      CALL #s_TRS5_FB_HW_MTR_MS (
           i_CMD_Send_Stat          := #i_Send_Statistics,
           i_Event_DB               := "DB_Event_Section",
           i_Available_IO           := #i_IO_Available,
           i_IO_MS_Automatic_Mode   := TRUE,
           i_IO_NOT_THO             := #i_TRS5_IO_NOT_THO,
           i_CMD_Reset              := #i_CMD_Reset,
           i_CMD_Req_Motor_Forward  := #s_TRS5_Req_MTR_Run,
           i_CMD_Manual_Mode        := #i_Command.Manual,
           i_CMD_Manual_Run         := #i_Command.Man_TRS5_Start,
           o_IO_MTR                 := #o_TRS5_IO_MTR,
           o_ST_THO                 := #s_TRS5_ST_THO);

NETWORK
TITLE =PA: Tracking report TRS5
//Case 1: SCZ01 in position Straight
//- Direction Taken 2, Decision Level 8 with ID of TRS5
//
//Case 2: SCZ01 in position Down
//- Direction Taken 2, Decision Level 3 with ID of TRS2
//- Direction From 1, Decision Level 3 with ID of TRS5
//
//In position down.
//When the item entering the downstream section a message "Direction From" with
//value "1" is sent to HLC with The ID of the TRS5.
      NOP   0;
// Tracking report Direction to: 2 (Item goes from up to down) second message
      A     #s_TRS5_Send_Track_Report;
      FN    #s_TRS5_FN_Send_Track_Rep;
      JCN   PA06;

      A     #s_SWS1_ST_Down;
      JCN   PA04;

// Create reply route record if not existing
      CALL "FC_Read_Int_Record" (
           i_Record_Number          := #s_TRS5_Fnd_LNK,
           i_P_INT_Record           := "DB_UDT_LNK_Record".Rep_Route,
           i_DB                     := "DB_LNK_List",
           i_DB_Event_Num           := #t_DB_Event_Section_Num,
           o_INT                    := #s_TRS5_Rep_Route_Record);

      L     #s_TRS5_Rep_Route_Record;
      L     0;
      <=I   ;
      JCN   PA01;

      CALL "FC_Generator_LNK" (
           i_LNK                    := #s_TRS5_Fnd_LNK,
           i_DB_List                := #t_DB_Nr_Route_List,
           i_Default_Record         := -1,
           i_DB_Event_Num           := #t_DB_Event_Section_Num,
           o_LNK                    := #s_TRS5_Rep_Route_Record);

      CALL "FC_Read_Int_Record" (
           i_Record_Number          := #s_TRS5_Fnd_LNK,
           i_P_INT_Record           := "DB_UDT_LNK_Record".Rep_Route,
           i_DB                     := "DB_LNK_List",
           i_DB_Event_Num           := #t_DB_Event_Section_Num,
           o_INT                    := #s_TRS5_Rep_Route_Record);

      CALL "FC_Read_Int_Record" (
           i_Record_Number          := #s_TRS5_Fnd_LNK,
           i_P_INT_Record           := "DB_UDT_LNK_Record".LIC,
           i_DB                     := "DB_LNK_List",
           i_DB_Event_Num           := #t_DB_Event_Section_Num,
           o_INT                    := #t_LIC);

      CALL "FC_Read_ANY_Record" (
           i_Record_Number          := #t_LIC,
           i_ANY_Data_Record        := "DB_UDT_LIC_Record".BIR,
           i_ANY_Data               := "DB_Outgoing_Msgs".TrackingReport.Body.BIR,
           i_DB                     := "DB_LIC_List",
           i_DB_Event_Num           := #t_DB_Event_Section_Num);

      CALL "FC_Write_ANY_Record" (
           i_Record_Number          := #s_TRS5_Rep_Route_Record,
           i_ANY_Data_Record        := "DB_UDT_Route_Record".BIR,
           i_ANY_Data               := "DB_Outgoing_Msgs".TrackingReport.Body.BIR,
           i_DB                     := "DB_Route_List",
           i_DB_Event_Num           := #t_DB_Event_Section_Num);

// Update tracking report message
PA01: CALL "FC_Write_ANY_Record" (
           i_Record_Number          := #s_TRS5_Rep_Route_Record,
           i_ANY_Data_Record        := "DB_UDT_Route_Record".SuccessDirection,
           i_ANY_Data               := "DB_Route_List".Rep_Route[0].SuccessDirection,
           i_DB                     := "DB_Route_List",
           i_DB_Event_Num           := #t_DB_Event_Section_Num);

      CALL "FC_Write_Int_Record" (
           i_Record_Number          := #s_TRS5_Rep_Route_Record,
           i_P_INT_Record           := "DB_UDT_Route_Record".SuccessDirection.DirectionFrom,
           i_DB                     := "DB_Route_List",
           i_INT                    := 0,
           i_DB_Event_Num           := #t_DB_Event_Section_Num);

      CALL "FC_Write_Int_Record" (
           i_Record_Number          := #s_TRS5_Rep_Route_Record,
           i_P_INT_Record           := "DB_UDT_Route_Record".SuccessDirection.DirectionTaken,
           i_DB                     := "DB_Route_List",
           i_INT                    := 2,
           i_DB_Event_Num           := #t_DB_Event_Section_Num);

      CALL "FC_Write_Int_Record" (
           i_Record_Number          := #s_TRS5_Rep_Route_Record,
           i_P_INT_Record           := "DB_UDT_Route_Record".SuccessDirection.DecisionLevel,
           i_DB                     := "DB_Route_List",
           i_INT                    := 5,
           i_DB_Event_Num           := #t_DB_Event_Section_Num);

// Write sort report
      CALL "FC_Write_Event" (
           i_Message_ID             := 1201,//Tracking Report = 1201
           i_Event_value            := #s_TRS5_Fnd_LNK,
           i_DB_Event_Num           := #t_DB_Event_Section_Num,
           o_Return_Value           := #t_RET_VAL_int);
      JU    PA06;


// Tracking report Direction to: 2 (Item goes straight)
PA04: A     #s_SWS1_ST_Straight;
      JCN   PA06;

// Create reply route record if not existing
      CALL "FC_Read_Int_Record" (
           i_Record_Number          := #s_TRS5_Fnd_LNK,
           i_P_INT_Record           := "DB_UDT_LNK_Record".Rep_Route,
           i_DB                     := "DB_LNK_List",
           i_DB_Event_Num           := #t_DB_Event_Section_Num,
           o_INT                    := #s_TRS5_Rep_Route_Record);

      L     #s_TRS5_Rep_Route_Record;
      L     0;
      <=I   ;
      JCN   PA05;

      CALL "FC_Generator_LNK" (
           i_LNK                    := #s_TRS5_Fnd_LNK,
           i_DB_List                := #t_DB_Nr_Route_List,
           i_Default_Record         := -1,
           i_DB_Event_Num           := #t_DB_Event_Section_Num,
           o_LNK                    := #s_TRS5_Rep_Route_Record);

      CALL "FC_Read_Int_Record" (
           i_Record_Number          := #s_TRS5_Fnd_LNK,
           i_P_INT_Record           := "DB_UDT_LNK_Record".Rep_Route,
           i_DB                     := "DB_LNK_List",
           i_DB_Event_Num           := #t_DB_Event_Section_Num,
           o_INT                    := #s_TRS5_Rep_Route_Record);

      CALL "FC_Read_Int_Record" (
           i_Record_Number          := #s_TRS5_Fnd_LNK,
           i_P_INT_Record           := "DB_UDT_LNK_Record".LIC,
           i_DB                     := "DB_LNK_List",
           i_DB_Event_Num           := #t_DB_Event_Section_Num,
           o_INT                    := #t_LIC);

      CALL "FC_Read_ANY_Record" (
           i_Record_Number          := #t_LIC,
           i_ANY_Data_Record        := "DB_UDT_LIC_Record".BIR,
           i_ANY_Data               := "DB_Outgoing_Msgs".TrackingReport.Body.BIR,
           i_DB                     := "DB_LIC_List",
           i_DB_Event_Num           := #t_DB_Event_Section_Num);

      CALL "FC_Write_ANY_Record" (
           i_Record_Number          := #s_TRS5_Rep_Route_Record,
           i_ANY_Data_Record        := "DB_UDT_Route_Record".BIR,
           i_ANY_Data               := "DB_Outgoing_Msgs".TrackingReport.Body.BIR,
           i_DB                     := "DB_Route_List",
           i_DB_Event_Num           := #t_DB_Event_Section_Num);

// Update tracking report message
PA05: CALL "FC_Write_ANY_Record" (
           i_Record_Number          := #s_TRS5_Rep_Route_Record,
           i_ANY_Data_Record        := "DB_UDT_Route_Record".SuccessDirection,
           i_ANY_Data               := "DB_Route_List".Rep_Route[0].SuccessDirection,
           i_DB                     := "DB_Route_List",
           i_DB_Event_Num           := #t_DB_Event_Section_Num);

      CALL "FC_Write_Int_Record" (
           i_Record_Number          := #s_TRS5_Rep_Route_Record,
           i_P_INT_Record           := "DB_UDT_Route_Record".SuccessDirection.DirectionFrom,
           i_DB                     := "DB_Route_List",
           i_INT                    := 0,
           i_DB_Event_Num           := #t_DB_Event_Section_Num);

      CALL "FC_Write_Int_Record" (
           i_Record_Number          := #s_TRS5_Rep_Route_Record,
           i_P_INT_Record           := "DB_UDT_Route_Record".SuccessDirection.DirectionTaken,
           i_DB                     := "DB_Route_List",
           i_INT                    := 1,
           i_DB_Event_Num           := #t_DB_Event_Section_Num);

      CALL "FC_Write_Int_Record" (
           i_Record_Number          := #s_TRS5_Rep_Route_Record,
           i_P_INT_Record           := "DB_UDT_Route_Record".SuccessDirection.DecisionLevel,
           i_DB                     := "DB_Route_List",
           i_INT                    := 5,
           i_DB_Event_Num           := #t_DB_Event_Section_Num);

// Write sort report
      CALL "FC_Write_Event" (
           i_Message_ID             := 1201,//Tracking Report = 1201
           i_Event_value            := #s_TRS5_Fnd_LNK,
           i_DB_Event_Num           := #t_DB_Event_Section_Num,
           o_Return_Value           := #t_RET_VAL_int);

PA06: CALL #s_TRS5_FB_DAT (
           i_ID_Section             := #i_TRS5_ID,
           i_DB_Event               := "DB_Event_Section",
           i_PLC_Log_FIFO_DB        := "DB_LOG_Event_FIFO",
           i_CFG_BPI_Log_Level      := "DB_Setting".common.External_Log_Level,
           i_CFG_PLC_Log_Level      := "DB_Setting".common.Internal_Log_Level,
           i_CFG_PLC_Log_Route_Msgs := TRUE,
           i_CFG_PLC_LOG_BPI_Stat   := FALSE,
           i_CFG_PLC_No_Msg_To_Rout := #i_CFG_PLC_No_Msg_To_Rout);

NETWORK
TITLE =QA: Data layer of SCZ01
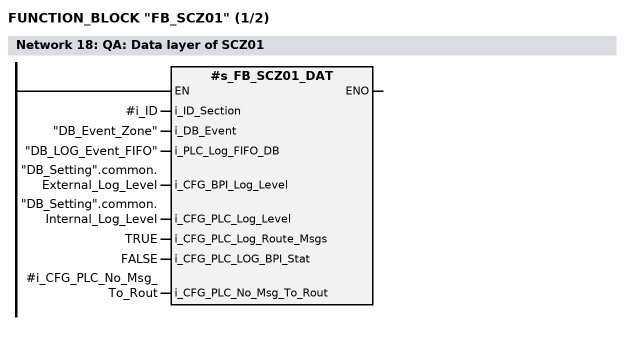

      CALL #s_FB_SCZ01_DAT (
           i_ID_Section             := #i_ID,
           i_DB_Event               := "DB_Event_Zone",
           i_PLC_Log_FIFO_DB        := "DB_LOG_Event_FIFO",
           i_CFG_BPI_Log_Level      := "DB_Setting".common.External_Log_Level,
           i_CFG_PLC_Log_Level      := "DB_Setting".common.Internal_Log_Level,
           i_CFG_PLC_Log_Route_Msgs := TRUE,
           i_CFG_PLC_LOG_BPI_Stat   := FALSE,
           i_CFG_PLC_No_Msg_To_Rout := #i_CFG_PLC_No_Msg_To_Rout);

NETWORK
TITLE =RA: Copy statistics, ready to restart and action active
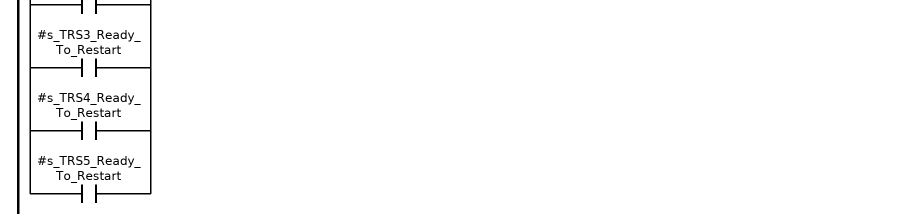

      A     #s_SWS1_ST_Up;
      =     #o_ST_Up;
      A     #s_SWS1_ST_Straight;
      =     #o_ST_Straight;
      A     #s_SWS1_ST_Down;
      =     #o_ST_Down;
      A     #s_ST_Fence_Opened;
      =     #o_ST_Fence_Opened;
      A     #s_ST_Gap_Blockage_Up;
      =     #o_ST_Gap_Blockage_Up;
      A     #s_ST_Gap_Blockage_Down;
      =     #o_ST_Gap_Blockage_Down;
      A     #s_ST_Gap_Switch_Up;
      =     #o_ST_Gap_Switch_Up;
      A     #s_ST_Gap_Switch_Down;
      =     #o_ST_Gap_Switch_Down;
      A     #s_SWS1_Mvdr_LS_Down;
      =     #o_SWS1_ST_LS_Limit_Down;
      A     #s_SWS1_Mvdr_LS_Up;
      =     #o_SWS1_ST_LS_Limit_Up;
      A     #s_SWS1_ST_Time_Out_Down;
      O     #s_SWS1_ST_Time_Out_Strgt;
      O     #s_SWS1_ST_Time_Out_Up;
      =     #o_SWS1_ST_Move_Time_Out;

// Mode
      A     #i_Command.Manual;
      =     #o_ST_Manual;
      A     #i_Command.Auto_Redun_Up;
      =     #o_ST_Redundant_Up;
      A     #i_Command.Auto_Redun_Dn;
      =     #o_ST_Redundant_Down;
      A     #i_Command.SemiAuto_Fix_Up;
      =     #o_ST_Fixed_Up;
      A     #i_Command.SemiAuto_Fix_Dn;
      =     #o_ST_Fixed_Down;
      A     #i_Command.SemiAuto_Fix_St;
      =     #o_ST_Fixed_Straight;

// TRS 2
      A     #s_TRS2_ST_EOS_PEC_Blk;
      =     #o_TRS2_ST_EOS_PEC_Blk;
      A     #s_TRS2_ST_EOS_PEC_Miss;
      =     #o_TRS2_ST_EOS_PEC_Miss;
      A     #s_TRS2_ST_THO;
      =     #o_TRS2_ST_THO;
      A     #s_TRS2_ST_PPI_Err;
      =     #o_TRS2_ST_PPI_Err;
      A     #s_TRS2_ST_Items;
      =     #o_TRS2_ST_Items;
      A     #s_TRS2_ST_Running;
      =     #o_TRS2_ST_Running;

// TRS 3
      A     #s_TRS3_ST_EOS_PEC_Blk;
      =     #o_TRS3_ST_EOS_PEC_Blk;
      A     #s_TRS3_ST_EOS_PEC_Miss;
      =     #o_TRS3_ST_EOS_PEC_Miss;
      A     #s_TRS3_ST_THO;
      =     #o_TRS3_ST_THO;
      A     #s_TRS3_ST_PPI_Err;
      =     #o_TRS3_ST_PPI_Err;

// TRS 4
      A     #s_TRS4_ST_EOS_PEC_Blk;
      =     #o_TRS4_ST_EOS_PEC_Blk;
      A     #s_TRS4_ST_EOS_PEC_Miss;
      =     #o_TRS4_ST_EOS_PEC_Miss;
      A     #s_TRS4_ST_THO;
      =     #o_TRS4_ST_THO;
      A     #s_TRS4_ST_PPI_Err;
      =     #o_TRS4_ST_PPI_Err;
      A     #s_TRS4_ST_Items;
      =     #o_TRS4_ST_Items;
      A     #s_TRS4_ST_Running;
      =     #o_TRS4_ST_Running;

// TRS 5
      A     #s_TRS5_ST_EOS_PEC_Blk;
      =     #o_TRS5_ST_EOS_PEC_Blk;
      A     #s_TRS5_ST_EOS_PEC_Miss;
      =     #o_TRS5_ST_EOS_PEC_Miss;
      A     #s_TRS5_ST_THO;
      =     #o_TRS5_ST_THO;
      A     #s_TRS5_ST_PPI_Err;
      =     #o_TRS5_ST_PPI_Err;

// Action active
      A     #o_SWS1_ST_Running;
      AN    #s_SWS1_Ext_Req_Stop;
      AN    #s_TRS2_Req_Stop;
      AN    #s_TRS3_Req_Stop;
      AN    #s_TRS4_Req_Stop;
      AN    #s_TRS5_Req_Stop;
      =     #o_Action_Active;

// Ready to start
      A     #s_SWS1_Ready_To_Restart;
      O     #s_TRS2_Ready_To_Restart;
      O     #s_TRS3_Ready_To_Restart;
      O     #s_TRS4_Ready_To_Restart;
      O     #s_TRS5_Ready_To_Restart;
      =     #o_Ready_To_Restart;

END_FUNCTION_BLOCK

